Fanuc KAREL source: port_OPOUT.kl

PROGRAM TP
%NOLOCKGROUP
VAR
 x: BOOLEAN
BEGIN
 x = OPOUT[3]
END TP
